VAR_GLOBAL CONSTANT
	cusiMinAddedChilds: USINT := 1;
	cusiSectionBuffer_SIZE: USINT := 20;
	cMAX_JAM_SENSORS: USINT := 3;
END_VAR

(* stored: Version 1.1.0.1, ProductVersion 3.1.0.19
   GVL Const_MER: Id {57566f58-da9e-4f02-8195-399b566f3bcb} *)
